{attribute 'qualified_only'}
VAR_GLOBAL
	R1_S1_EL1008		AT %I* : ARRAY[0..7] OF BOOL;
END_VAR

(* stored: Version 1.1.0.1, ProductVersion 3.1.4024.12
   GVL IO: Id {e5dfb23d-4ed5-43a6-abf9-cd4e88b77745} *)
